# EPICS autosave request: iocBoot/obsolete/ioc13Galil_test/auto_settings.req
file "CARS_8_motor_settings.req",  P=$(P)

file "galil_motor_extras.req",     P=$(P), M=m1
file "galil_motor_extras.req",     P=$(P), M=m2
file "galil_motor_extras.req",     P=$(P), M=m3
file "galil_motor_extras.req",     P=$(P), M=m4
file "galil_motor_extras.req",     P=$(P), M=m5
file "galil_motor_extras.req",     P=$(P), M=m6
file "galil_motor_extras.req",     P=$(P), M=m7
file "galil_motor_extras.req",     P=$(P), M=m8
